(* CoDeSys 2.3 export: ST_SENSOR_KG.EXP *)

(* Data type *)
TYPE ST_SENSOR_KG :
STRUCT
	Name : STRING;

	Raw : REAL;
	Kg  : REAL;

	(*Calib*)
	Cal_K : REAL;
	Cal_C : REAL;

END_STRUCT
END_TYPE
